// TIA Portal V20 export
TYPE "zp_Tool_Data"
// stored: Access Published, Namespace CITI_Logic
   STRUCT
      ToolPocketOrStaNumber : Int;
      SerialNumber : DInt;
      ToolTypeOrGroup : String[12];
      MaximumToolLife : DInt;
      ToolLifeWarningLimit : DInt;
      ToolCyclesUsed : DInt;
   END_STRUCT;
END_TYPE
